FUNCTION_BLOCK FB_LongTransfer IMPLEMENTS I_ControlScheme
VAR_INPUT
END_VAR
VAR_OUTPUT
END_VAR
VAR
	fbDecline	: FB_DeclineMdrConveyer;
	fbLongStraight1		: FB_LsMdrConveyer;
	fbLongStraight2		: FB_LsMdrConveyer;
	nState: INT;
END_VAR
VAR_IN_OUT
	Axis1	:	EP7402_REF;
	Axis2	:	EP7402_REF;
	Axis3	:	EP7402_REF;
END_VAR

CASE nState OF
0:
	//TODO:Assign Axes
	nState :=1;
1: 
	fbLongStraight1.Start();
	fbLongStraight2.Start();
	fbDecline.Start();
	
	
	
2:
	fbLongStraight1.Execute();
	fbLongStraight2.Execute();
	fbDecline.Execute();
	

	nState := 3;
3:
	//TO-DO call Stop methods
	nState := 4;
4:
	//TODO: call Reset methods
END_CASE

END_FUNCTION_BLOCK

(* stored: Version 1.1.0.1, ProductVersion 3.1.4024.6
   POU FB_LongTransfer: Id {48ec9a18-fd00-46eb-9f61-e8dc50e77b27}, SpecialFunc None *)
